{attribute 'GeneratedUsingTerminal: DL-EC1A-0000'}
{attribute addProperty BoxType "DL-EC1A-0000"}
{attribute addProperty Id "WcStateAT %I*BOOL1InputToggleAT %I*BOOL1"}
{attribute addProperty CRC "2425479403"}
{attribute addProperty Size "2"}
TYPE
    WcState_9091E0EB :
    STRUCT
        {attribute addProperty Name "WcState"}
        WcState AT %I* : BOOL;
        {attribute addProperty Name "InputToggle"}
        InputToggle AT %I* : BOOL;
    END_STRUCT
END_TYPE

(* stored: Version 1.1.0.1, ProductVersion 3.1.4024.12
   DUT WcState_9091E0EB: Id {6fc2218b-ded4-0439-33e3-a3e02d9706b0} *)
